FUNCTION F_CarbideShutterEnable : BOOL
VAR_INPUT
END_VAR
VAR_IN_OUT CONSTANT
	stErrors : ST_ErrorStates;
END_VAR
VAR
END_VAR

F_CarbideShutterEnable := FALSE;

// Close carbide shutter if there is a hardware failure
IF stErrors.bHardwareFailure THEN
	RETURN;
END_IF

// Close carbide shutter if leak in OPCPA with carbide on or if there is a leak under the table
IF stErrors.bLeakOpcpaCarbideOn OR stErrors.bLeakUnderTable THEN
	RETURN;
END_IF

F_CarbideShutterEnable := TRUE;

END_FUNCTION

(* stored: Version 1.1.0.1, ProductVersion 3.1.4020.14
   POU F_CarbideShutterEnable: Id {6b2b070e-0295-4d27-a821-90f06b1926e9}, SpecialFunc None *)
